FUNCTION_BLOCK FB_LamparaAsignada_ST
VAR_INPUT
END_VAR
VAR_OUTPUT
END_VAR
VAR
    Lampara AT %Q*: BOOL;
    Pulsador AT %I*: BOOL;
END_VAR

Lampara := Pulsador;

END_FUNCTION_BLOCK

(* stored: Version 1.1.0.1, ProductVersion 3.1.4024.15
   POU FB_LamparaAsignada_ST: Id {cb0c5f12-56d6-46fd-b76b-40c9b1cfc97a}, SpecialFunc None *)
